// TIA Portal V17 export
// export: Created 2023-12-22T15:04:41.1815783Z, ExportSetting WithDefaults, DisplayName Totally Integrated Automation Portal, DisplayVersion V17, DisplayName TIA Portal Openness, DisplayVersion V17, DisplayName TIA Portal Version Control Interface, DisplayVersion V17, DisplayName STEP 7 Professional, DisplayVersion V17, DisplayName STEP 7 Safety, DisplayVersion V17, DisplayName WinCC Advanced, DisplayVersion V17
FUNCTION_BLOCK "Motors"   // FB240, LAD
{ S7_Optimized_Access := 'FALSE' }
VERSION : 0.1
// stored: AutoNumber false, IsIECCheckEnabled false, SetENOAutomatically false, UDAEnableTagReadback false
   VAR DB_SPECIFIC
      Time_DTL { S7_SetPoint := 'True'} : DTL;
   END_VAR
BEGIN

REGION Network 1: Мешалки
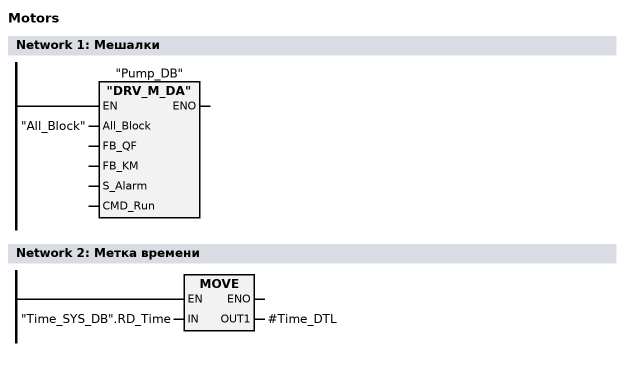
   RUNG wire#powerrail
      "Pump_DB"(All_Block := "All_Block", FB_QF :=, FB_KM :=, S_Alarm :=, CMD_Run :=)
   END_RUNG
   // the same network as SCL:
   "Pump_DB"(All_Block := "All_Block");   // "DRV_M_DA"
END_REGION

REGION Network 2: Метка времени
   RUNG wire#powerrail
      Move(in := "Time_SYS_DB".RD_Time, out1 => #Time_DTL)
   END_RUNG
   // the same network as SCL:
   #Time_DTL := "Time_SYS_DB".RD_Time;
END_REGION
END_FUNCTION_BLOCK
